TYPE ST_Device :
STRUCT
	sDeviceName : STRING;
	nDeviceValue : INT;
END_STRUCT
END_TYPE

(* stored: Version 1.1.0.1, ProductVersion 3.1.4024.16
   DUT ST_Device: Id {9b8be032-3a69-41ec-a235-fd01e121cedb} *)
